// TIA Portal V18 export
FUNCTION_BLOCK "MES_CHeck"   // FB111, LAD
{ S7_Optimized_Access := 'TRUE' }
VERSION : 0.1
// stored: AutoNumber false, IsIECCheckEnabled false, IsRetainMemResEnabled false, MemoryReserve 100, SetENOAutomatically false, UDAEnableTagReadback false
   VAR
      Station_1 : "MES Check_fb";   // *
      Station_2 : "MES Check_fb";   // *
      Station_3 : "MES Check_fb";   // *
      Station_4 : "MES Check_fb";   // *
      Station_5 : "MES Check_fb";   // *
      Station_6 : "MES Check_fb";   // *
      Station_7 : "MES Check_fb";   // *
      Station_8 : "MES Check_fb";   // *
   END_VAR
BEGIN

REGION Network 1: Station_1 shaft_1
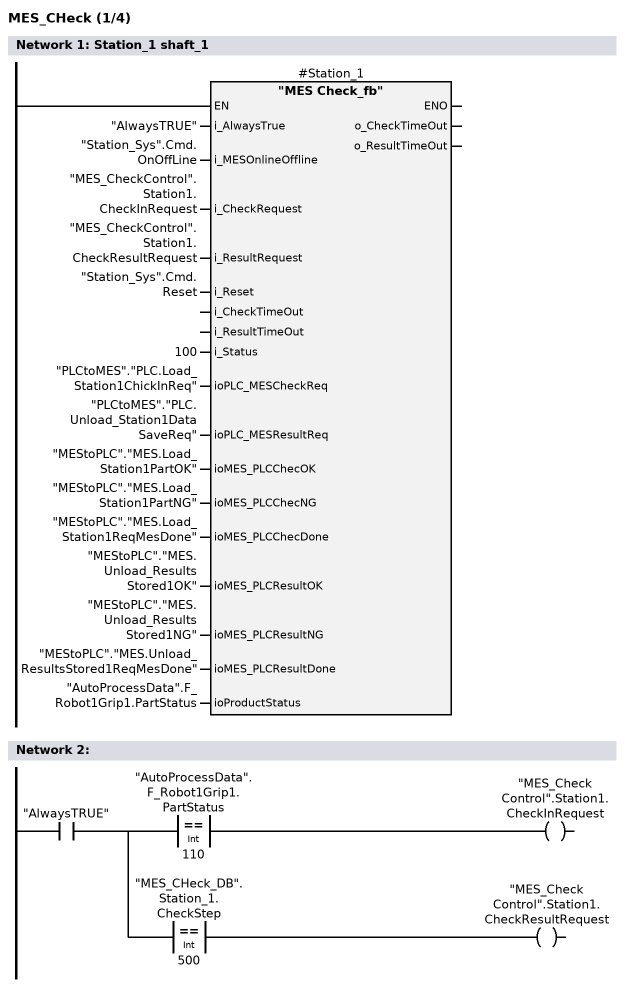
   RUNG wire#powerrail
      #Station_1(i_AlwaysTrue := "AlwaysTRUE", i_MESOnlineOffline := "Station_Sys".Cmd.OnOffLine, i_CheckRequest := "MES_CheckControl".Station1.CheckInRequest, i_ResultRequest := "MES_CheckControl".Station1.CheckResultRequest, i_Reset := "Station_Sys".Cmd.Reset, i_CheckTimeOut :=, i_ResultTimeOut :=, i_Status := 100, ioPLC_MESCheckReq := "PLCtoMES"."PLC.Load_Station1ChickInReq", ioPLC_MESResultReq := "PLCtoMES"."PLC.Unload_Station1DataSaveReq", ioMES_PLCChecOK := "MEStoPLC"."MES.Load_Station1PartOK", ioMES_PLCChecNG := "MEStoPLC"."MES.Load_Station1PartNG", ioMES_PLCChecDone := "MEStoPLC"."MES.Load_Station1ReqMesDone", ioMES_PLCResultOK := "MEStoPLC"."MES.Unload_ResultsStored1OK", ioMES_PLCResultNG := "MEStoPLC"."MES.Unload_ResultsStored1NG", ioMES_PLCResultDone := "MEStoPLC"."MES.Unload_ResultsStored1ReqMesDone", ioProductStatus := "AutoProcessData".F_Robot1Grip1.PartStatus, o_CheckTimeOut =>, o_ResultTimeOut =>)
   END_RUNG
   // the same network as SCL:
   #Station_1(i_AlwaysTrue := "AlwaysTRUE",   // "MES Check_fb"
              i_MESOnlineOffline := "Station_Sys".Cmd.OnOffLine,
              i_CheckRequest := "MES_CheckControl".Station1.CheckInRequest,
              i_ResultRequest := "MES_CheckControl".Station1.CheckResultRequest,
              i_Reset := "Station_Sys".Cmd.Reset,
              i_Status := 100,
              ioPLC_MESCheckReq := "PLCtoMES"."PLC.Load_Station1ChickInReq",
              ioPLC_MESResultReq := "PLCtoMES"."PLC.Unload_Station1DataSaveReq",
              ioMES_PLCChecOK := "MEStoPLC"."MES.Load_Station1PartOK",
              ioMES_PLCChecNG := "MEStoPLC"."MES.Load_Station1PartNG",
              ioMES_PLCChecDone := "MEStoPLC"."MES.Load_Station1ReqMesDone",
              ioMES_PLCResultOK := "MEStoPLC"."MES.Unload_ResultsStored1OK",
              ioMES_PLCResultNG := "MEStoPLC"."MES.Unload_ResultsStored1NG",
              ioMES_PLCResultDone := "MEStoPLC"."MES.Unload_ResultsStored1ReqMesDone",
              ioProductStatus := "AutoProcessData".F_Robot1Grip1.PartStatus);
END_REGION

REGION Network 2
   RUNG wire#powerrail
      Contact( "AlwaysTRUE" )
      wire#w1
      { S7_Templates := "SrcType := Int" } EQ_Contact(in1 := "AutoProcessData".F_Robot1Grip1.PartStatus, in2 := 110)
      Coil( "MES_CheckControl".Station1.CheckInRequest )
   END_RUNG
   RUNG wire#w1
      { S7_Templates := "SrcType := Int" } EQ_Contact(in1 := "MES_CHeck_DB".Station_1.CheckStep, in2 := 500)
      Coil( "MES_CheckControl".Station1.CheckResultRequest )
   END_RUNG
   // the same network as SCL:
   "MES_CheckControl".Station1.CheckInRequest := "AlwaysTRUE" AND ("AutoProcessData".F_Robot1Grip1.PartStatus = 110);
   "MES_CheckControl".Station1.CheckResultRequest := "AlwaysTRUE" AND ("MES_CHeck_DB".Station_1.CheckStep = 500);
END_REGION

REGION Network 3: Station_2 Ring_1
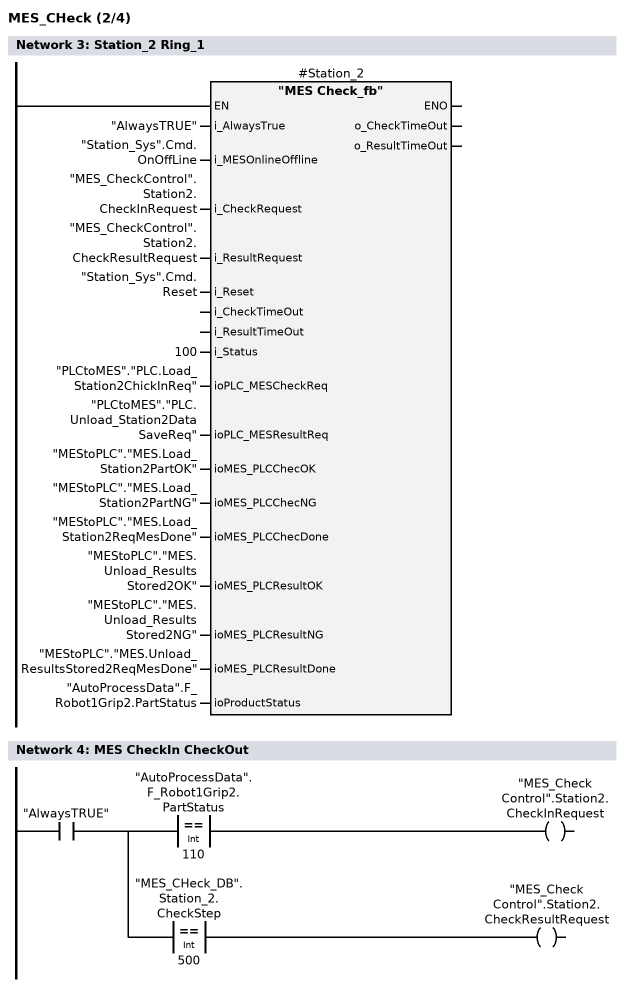
   RUNG wire#powerrail
      #Station_2(i_AlwaysTrue := "AlwaysTRUE", i_MESOnlineOffline := "Station_Sys".Cmd.OnOffLine, i_CheckRequest := "MES_CheckControl".Station2.CheckInRequest, i_ResultRequest := "MES_CheckControl".Station2.CheckResultRequest, i_Reset := "Station_Sys".Cmd.Reset, i_CheckTimeOut :=, i_ResultTimeOut :=, i_Status := 100, ioPLC_MESCheckReq := "PLCtoMES"."PLC.Load_Station2ChickInReq", ioPLC_MESResultReq := "PLCtoMES"."PLC.Unload_Station2DataSaveReq", ioMES_PLCChecOK := "MEStoPLC"."MES.Load_Station2PartOK", ioMES_PLCChecNG := "MEStoPLC"."MES.Load_Station2PartNG", ioMES_PLCChecDone := "MEStoPLC"."MES.Load_Station2ReqMesDone", ioMES_PLCResultOK := "MEStoPLC"."MES.Unload_ResultsStored2OK", ioMES_PLCResultNG := "MEStoPLC"."MES.Unload_ResultsStored2NG", ioMES_PLCResultDone := "MEStoPLC"."MES.Unload_ResultsStored2ReqMesDone", ioProductStatus := "AutoProcessData".F_Robot1Grip2.PartStatus, o_CheckTimeOut =>, o_ResultTimeOut =>)
   END_RUNG
   // the same network as SCL:
   #Station_2(i_AlwaysTrue := "AlwaysTRUE",   // "MES Check_fb"
              i_MESOnlineOffline := "Station_Sys".Cmd.OnOffLine,
              i_CheckRequest := "MES_CheckControl".Station2.CheckInRequest,
              i_ResultRequest := "MES_CheckControl".Station2.CheckResultRequest,
              i_Reset := "Station_Sys".Cmd.Reset,
              i_Status := 100,
              ioPLC_MESCheckReq := "PLCtoMES"."PLC.Load_Station2ChickInReq",
              ioPLC_MESResultReq := "PLCtoMES"."PLC.Unload_Station2DataSaveReq",
              ioMES_PLCChecOK := "MEStoPLC"."MES.Load_Station2PartOK",
              ioMES_PLCChecNG := "MEStoPLC"."MES.Load_Station2PartNG",
              ioMES_PLCChecDone := "MEStoPLC"."MES.Load_Station2ReqMesDone",
              ioMES_PLCResultOK := "MEStoPLC"."MES.Unload_ResultsStored2OK",
              ioMES_PLCResultNG := "MEStoPLC"."MES.Unload_ResultsStored2NG",
              ioMES_PLCResultDone := "MEStoPLC"."MES.Unload_ResultsStored2ReqMesDone",
              ioProductStatus := "AutoProcessData".F_Robot1Grip2.PartStatus);
END_REGION

REGION Network 4: MES CheckIn CheckOut
   RUNG wire#powerrail
      Contact( "AlwaysTRUE" )
      wire#w1
      { S7_Templates := "SrcType := Int" } EQ_Contact(in1 := "AutoProcessData".F_Robot1Grip2.PartStatus, in2 := 110)
      Coil( "MES_CheckControl".Station2.CheckInRequest )
   END_RUNG
   RUNG wire#w1
      { S7_Templates := "SrcType := Int" } EQ_Contact(in1 := "MES_CHeck_DB".Station_2.CheckStep, in2 := 500)
      Coil( "MES_CheckControl".Station2.CheckResultRequest )
   END_RUNG
   // the same network as SCL:
   "MES_CheckControl".Station2.CheckInRequest := "AlwaysTRUE" AND ("AutoProcessData".F_Robot1Grip2.PartStatus = 110);
   "MES_CheckControl".Station2.CheckResultRequest := "AlwaysTRUE" AND ("MES_CHeck_DB".Station_2.CheckStep = 500);
END_REGION

REGION Network 5: Station_4 Magnet
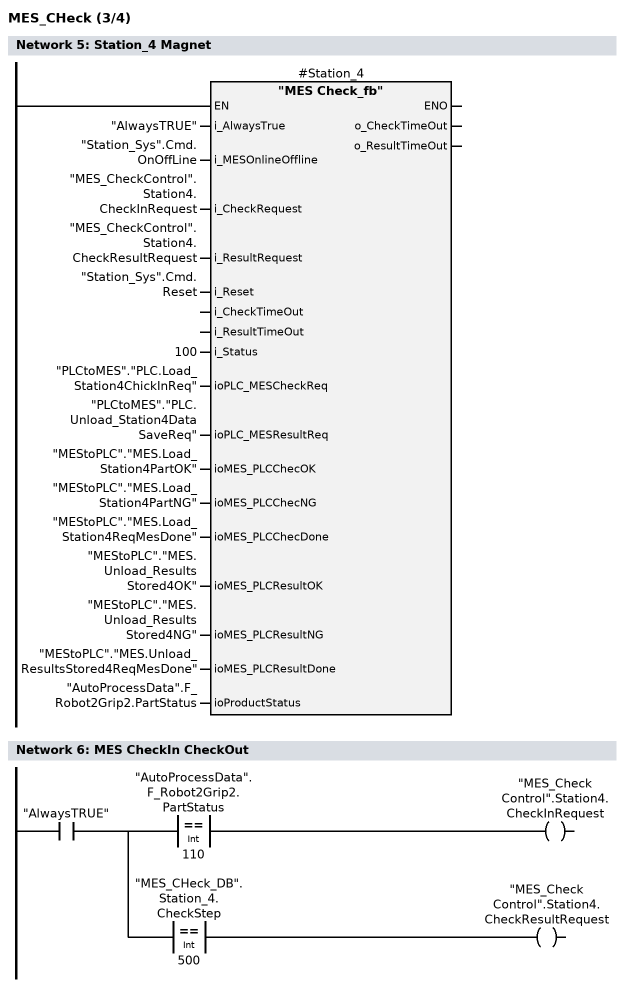
   RUNG wire#powerrail
      #Station_4(i_AlwaysTrue := "AlwaysTRUE", i_MESOnlineOffline := "Station_Sys".Cmd.OnOffLine, i_CheckRequest := "MES_CheckControl".Station4.CheckInRequest, i_ResultRequest := "MES_CheckControl".Station4.CheckResultRequest, i_Reset := "Station_Sys".Cmd.Reset, i_CheckTimeOut :=, i_ResultTimeOut :=, i_Status := 100, ioPLC_MESCheckReq := "PLCtoMES"."PLC.Load_Station4ChickInReq", ioPLC_MESResultReq := "PLCtoMES"."PLC.Unload_Station4DataSaveReq", ioMES_PLCChecOK := "MEStoPLC"."MES.Load_Station4PartOK", ioMES_PLCChecNG := "MEStoPLC"."MES.Load_Station4PartNG", ioMES_PLCChecDone := "MEStoPLC"."MES.Load_Station4ReqMesDone", ioMES_PLCResultOK := "MEStoPLC"."MES.Unload_ResultsStored4OK", ioMES_PLCResultNG := "MEStoPLC"."MES.Unload_ResultsStored4NG", ioMES_PLCResultDone := "MEStoPLC"."MES.Unload_ResultsStored4ReqMesDone", ioProductStatus := "AutoProcessData".F_Robot2Grip2.PartStatus, o_CheckTimeOut =>, o_ResultTimeOut =>)
   END_RUNG
   // the same network as SCL:
   #Station_4(i_AlwaysTrue := "AlwaysTRUE",   // "MES Check_fb"
              i_MESOnlineOffline := "Station_Sys".Cmd.OnOffLine,
              i_CheckRequest := "MES_CheckControl".Station4.CheckInRequest,
              i_ResultRequest := "MES_CheckControl".Station4.CheckResultRequest,
              i_Reset := "Station_Sys".Cmd.Reset,
              i_Status := 100,
              ioPLC_MESCheckReq := "PLCtoMES"."PLC.Load_Station4ChickInReq",
              ioPLC_MESResultReq := "PLCtoMES"."PLC.Unload_Station4DataSaveReq",
              ioMES_PLCChecOK := "MEStoPLC"."MES.Load_Station4PartOK",
              ioMES_PLCChecNG := "MEStoPLC"."MES.Load_Station4PartNG",
              ioMES_PLCChecDone := "MEStoPLC"."MES.Load_Station4ReqMesDone",
              ioMES_PLCResultOK := "MEStoPLC"."MES.Unload_ResultsStored4OK",
              ioMES_PLCResultNG := "MEStoPLC"."MES.Unload_ResultsStored4NG",
              ioMES_PLCResultDone := "MEStoPLC"."MES.Unload_ResultsStored4ReqMesDone",
              ioProductStatus := "AutoProcessData".F_Robot2Grip2.PartStatus);
END_REGION

REGION Network 6: MES CheckIn CheckOut
   RUNG wire#powerrail
      Contact( "AlwaysTRUE" )
      wire#w1
      { S7_Templates := "SrcType := Int" } EQ_Contact(in1 := "AutoProcessData".F_Robot2Grip2.PartStatus, in2 := 110)
      Coil( "MES_CheckControl".Station4.CheckInRequest )
   END_RUNG
   RUNG wire#w1
      { S7_Templates := "SrcType := Int" } EQ_Contact(in1 := "MES_CHeck_DB".Station_4.CheckStep, in2 := 500)
      Coil( "MES_CheckControl".Station4.CheckResultRequest )
   END_RUNG
   // the same network as SCL:
   "MES_CheckControl".Station4.CheckInRequest := "AlwaysTRUE" AND ("AutoProcessData".F_Robot2Grip2.PartStatus = 110);
   "MES_CheckControl".Station4.CheckResultRequest := "AlwaysTRUE" AND ("MES_CHeck_DB".Station_4.CheckStep = 500);
END_REGION

REGION Network 7: Station_6 Ring_2
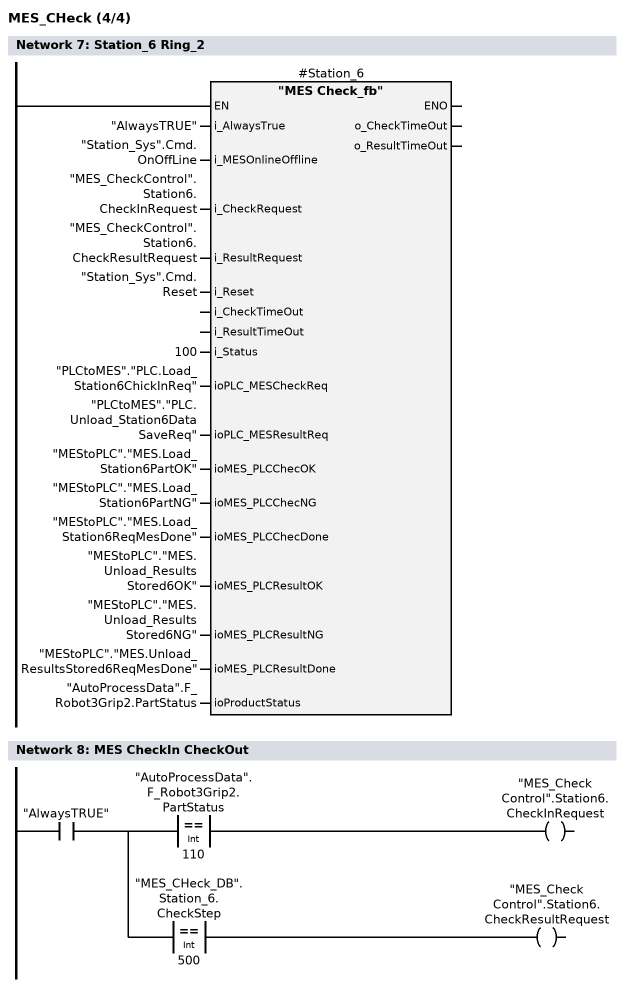
   RUNG wire#powerrail
      #Station_6(i_AlwaysTrue := "AlwaysTRUE", i_MESOnlineOffline := "Station_Sys".Cmd.OnOffLine, i_CheckRequest := "MES_CheckControl".Station6.CheckInRequest, i_ResultRequest := "MES_CheckControl".Station6.CheckResultRequest, i_Reset := "Station_Sys".Cmd.Reset, i_CheckTimeOut :=, i_ResultTimeOut :=, i_Status := 100, ioPLC_MESCheckReq := "PLCtoMES"."PLC.Load_Station6ChickInReq", ioPLC_MESResultReq := "PLCtoMES"."PLC.Unload_Station6DataSaveReq", ioMES_PLCChecOK := "MEStoPLC"."MES.Load_Station6PartOK", ioMES_PLCChecNG := "MEStoPLC"."MES.Load_Station6PartNG", ioMES_PLCChecDone := "MEStoPLC"."MES.Load_Station6ReqMesDone", ioMES_PLCResultOK := "MEStoPLC"."MES.Unload_ResultsStored6OK", ioMES_PLCResultNG := "MEStoPLC"."MES.Unload_ResultsStored6NG", ioMES_PLCResultDone := "MEStoPLC"."MES.Unload_ResultsStored6ReqMesDone", ioProductStatus := "AutoProcessData".F_Robot3Grip2.PartStatus, o_CheckTimeOut =>, o_ResultTimeOut =>)
   END_RUNG
   // the same network as SCL:
   #Station_6(i_AlwaysTrue := "AlwaysTRUE",   // "MES Check_fb"
              i_MESOnlineOffline := "Station_Sys".Cmd.OnOffLine,
              i_CheckRequest := "MES_CheckControl".Station6.CheckInRequest,
              i_ResultRequest := "MES_CheckControl".Station6.CheckResultRequest,
              i_Reset := "Station_Sys".Cmd.Reset,
              i_Status := 100,
              ioPLC_MESCheckReq := "PLCtoMES"."PLC.Load_Station6ChickInReq",
              ioPLC_MESResultReq := "PLCtoMES"."PLC.Unload_Station6DataSaveReq",
              ioMES_PLCChecOK := "MEStoPLC"."MES.Load_Station6PartOK",
              ioMES_PLCChecNG := "MEStoPLC"."MES.Load_Station6PartNG",
              ioMES_PLCChecDone := "MEStoPLC"."MES.Load_Station6ReqMesDone",
              ioMES_PLCResultOK := "MEStoPLC"."MES.Unload_ResultsStored6OK",
              ioMES_PLCResultNG := "MEStoPLC"."MES.Unload_ResultsStored6NG",
              ioMES_PLCResultDone := "MEStoPLC"."MES.Unload_ResultsStored6ReqMesDone",
              ioProductStatus := "AutoProcessData".F_Robot3Grip2.PartStatus);
END_REGION

REGION Network 8: MES CheckIn CheckOut
   RUNG wire#powerrail
      Contact( "AlwaysTRUE" )
      wire#w1
      { S7_Templates := "SrcType := Int" } EQ_Contact(in1 := "AutoProcessData".F_Robot3Grip2.PartStatus, in2 := 110)
      Coil( "MES_CheckControl".Station6.CheckInRequest )
   END_RUNG
   RUNG wire#w1
      { S7_Templates := "SrcType := Int" } EQ_Contact(in1 := "MES_CHeck_DB".Station_6.CheckStep, in2 := 500)
      Coil( "MES_CheckControl".Station6.CheckResultRequest )
   END_RUNG
   // the same network as SCL:
   "MES_CheckControl".Station6.CheckInRequest := "AlwaysTRUE" AND ("AutoProcessData".F_Robot3Grip2.PartStatus = 110);
   "MES_CheckControl".Station6.CheckResultRequest := "AlwaysTRUE" AND ("MES_CHeck_DB".Station_6.CheckStep = 500);
END_REGION
END_FUNCTION_BLOCK
